FUNCTION TryConvert_WORD_TO_LINT : BOOL
VAR_INPUT
	in : WORD;
	out : REFERENCE TO LINT;
END_VAR

out := WORD_TO_LINT(in);
TryConvert_WORD_TO_LINT := TRUE;

END_FUNCTION

(* stored: Version 1.1.0.1, ProductVersion 3.1.4024.12
   POU TryConvert_WORD_TO_LINT: Id {7ff920f8-6f55-498a-b663-3c273ebd8b6b}, SpecialFunc None *)
